{attribute 'GeneratedUsingTerminal: EP9224-0023-0016'}
{attribute addProperty BoxType "EP9224-0023-0016"}
{attribute addProperty Id "DPO_Inputs_Channel_1AT %I*DPO_Inputs_Channel_F87663B815DPO_Inputs_Channel_2AT %I*DPO_Inputs_Channel_F87663B815DPO_Inputs_Channel_3AT %I*DPO_Inputs_Channel_F87663B815DPO_Inputs_Channel_4AT %I*DPO_Inputs_Channel_F87663B815DPO_Inputs_DeviceAT %I*DPO_Inputs_Device_99241EEA22DPO_Outputs_Channel_1AT %Q*DPO_Outputs_Channel_A459B36C4DPO_Outputs_Channel_2AT %Q*DPO_Outputs_Channel_A459B36C4DPO_Outputs_Channel_3AT %Q*DPO_Outputs_Channel_A459B36C4DPO_Outputs_Channel_4AT %Q*DPO_Outputs_Channel_A459B36C4DPO_Outputs_DeviceAT %Q*DPO_Outputs_Device_B673A3372WcStateAT %I*WcState_9091E0EB2InfoDataAT %I*InfoData_94A18F5E2"}
{attribute addProperty CRC "512360230"}
{attribute addProperty Size "104"}
TYPE EP9224_1E89FF26 EXTENDS EtcSlaveTerminalBase_947E5A46 :
STRUCT
	{attribute addProperty Name "DPO_Inputs_Channel_1"}
	DPO_Inputs_Channel_1 : DPO_Inputs_Channel_F87663B8;
	{attribute addProperty Name "DPO_Inputs_Channel_2"}
	DPO_Inputs_Channel_2 : DPO_Inputs_Channel_F87663B8;
	{attribute addProperty Name "DPO_Inputs_Channel_3"}
	DPO_Inputs_Channel_3 : DPO_Inputs_Channel_F87663B8;
	{attribute addProperty Name "DPO_Inputs_Channel_4"}
	DPO_Inputs_Channel_4 : DPO_Inputs_Channel_F87663B8;
	{attribute addProperty Name "DPO_Inputs_Device"}
	DPO_Inputs_Device : DPO_Inputs_Device_99241EEA;
	{attribute addProperty Name "DPO_Outputs_Channel_1"}
	DPO_Outputs_Channel_1 : DPO_Outputs_Channel_A459B36C;
	{attribute addProperty Name "DPO_Outputs_Channel_2"}
	DPO_Outputs_Channel_2 : DPO_Outputs_Channel_A459B36C;
	{attribute addProperty Name "DPO_Outputs_Channel_3"}
	DPO_Outputs_Channel_3 : DPO_Outputs_Channel_A459B36C;
	{attribute addProperty Name "DPO_Outputs_Channel_4"}
	DPO_Outputs_Channel_4 : DPO_Outputs_Channel_A459B36C;
	{attribute addProperty Name "DPO_Outputs_Device"}
	DPO_Outputs_Device : DPO_Outputs_Device_B673A337;
	{attribute addProperty Name "WcState"}
	WcState : WcState_9091E0EB;
	{attribute addProperty Name "InfoData"}
	InfoData : InfoData_94A18F5E;
END_STRUCT
END_TYPE

(* stored: Version 1.2.0.0, ProductVersion 3.1.4024.9
   DUT EP9224_1E89FF26: Id {5ec0c02e-f33e-405f-87bd-ab93568617ad} *)
